(* IEC 61131-3 sources: horner-cscape-mcp/artifacts/projects/FailAudit_POU_MissingSemicolon/pous, 1 file *)

(* ---- POU_MissingSemicolon.st ---- *)
PROGRAM POU_MissingSemicolon
VAR
    BatchCount : INT := 10;
END_VAR
BatchCount := 42
END_PROGRAM
